// TIA Portal project "2022.06.10_多路模拟输入输出" (V17)

(* hardware
DEVICE "S7-1200 station_1"  S7-1200 Station
   slot 0: "Rack_0"  S7-1200 Rack  Rack  V1.0
   slot 1: "PLC_1"  CPU 1212C DC/DC/DC  6ES7 212-1AE40-0XB0  V4.5
   slot 2: "AI 4x13BIT/AQ 2x14BIT_1"  SM 1234 AI4/AQ2  6ES7 234-4HE30-0XB0  V1.0
*)

// ===== PLC "PLC_1"  CPU 1212C DC/DC/DC =====

VAR_GLOBAL   // PLC tag table "默认变量表"
   "所需频率" AT %IW96 : Word;
   "百分比" AT %MD40 : DWord;
   "模拟量输出通道" AT %MD44 : UDInt;
   "所需频率(1)" AT %MD0 : Real;
   "压力2模拟输入通道" AT %IW100 : Int;
   "压力2" AT %MD4 : Real;
END_VAR

FUNCTION "模拟量输入" : Void   // FC1, LAD
{ S7_Optimized_Access := 'TRUE' }
VERSION : 0.1
   VAR_INPUT
      模拟量输入上限 : Int;
      模拟量输入下限 : Int;
      工程之上限 : Real;
      工程值下限 : Real;
      模拟量输入值 : Int;
   END_VAR
   VAR_OUTPUT
      实际工程值 : Real;
   END_VAR
   VAR_TEMP
      百分比 : Bool;
   END_VAR
BEGIN

REGION Network 1
   // out只是中转，用temp
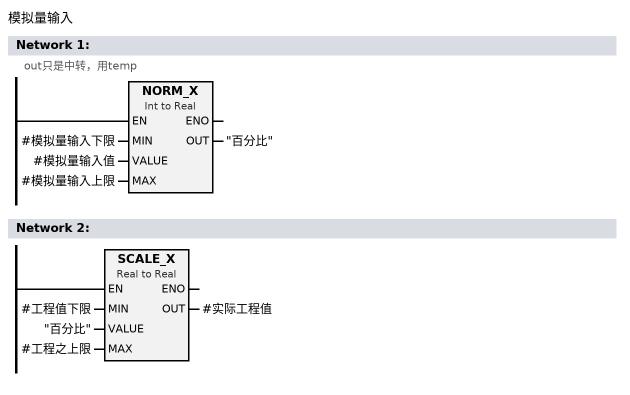
   RUNG wire#powerrail
      { S7_Templates := "[SrcType := Int, DestType := Real]" } Normalize(min := #模拟量输入下限, value := #模拟量输入值, max := #模拟量输入上限, out => "百分比")
   END_RUNG
   // the same network as SCL:
   "百分比" := NORM_X(MIN := #模拟量输入下限, VALUE := #模拟量输入值, MAX := #模拟量输入上限);
END_REGION

REGION Network 2
   RUNG wire#powerrail
      { S7_Templates := "[SrcType := Real, DestType := Real]" } Scale(min := #工程值下限, value := "百分比", max := #工程之上限, out => #实际工程值)
   END_RUNG
   // the same network as SCL:
   #实际工程值 := SCALE_X(MIN := #工程值下限, VALUE := "百分比", MAX := #工程之上限);
END_REGION
END_FUNCTION

FUNCTION "多路模拟量" : Void   // FC2, LAD
{ S7_Optimized_Access := 'TRUE' }
VERSION : 0.1
BEGIN

REGION Network 1
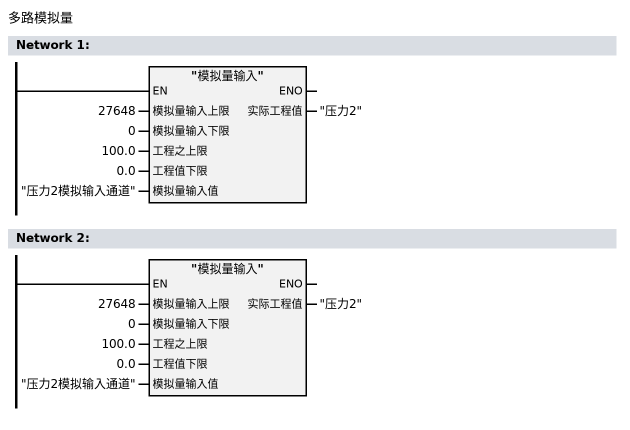
   RUNG wire#powerrail
      "模拟量输入"(模拟量输入上限 := 27648, 模拟量输入下限 := 0, 工程之上限 := 100.0, 工程值下限 := 0.0, 模拟量输入值 := "压力2模拟输入通道", 实际工程值 => "压力2")
   END_RUNG
   // the same network as SCL:
   "模拟量输入"(模拟量输入上限 := 27648, 模拟量输入下限 := 0, 工程之上限 := 100.0, 工程值下限 := 0.0, 模拟量输入值 := "压力2模拟输入通道", 实际工程值 => "压力2");
END_REGION

REGION Network 2
   RUNG wire#powerrail
      "模拟量输入"(模拟量输入上限 := 27648, 模拟量输入下限 := 0, 工程之上限 := 100.0, 工程值下限 := 0.0, 模拟量输入值 := "压力2模拟输入通道", 实际工程值 => "压力2")
   END_RUNG
   // the same network as SCL:
   "模拟量输入"(模拟量输入上限 := 27648, 模拟量输入下限 := 0, 工程之上限 := 100.0, 工程值下限 := 0.0, 模拟量输入值 := "压力2模拟输入通道", 实际工程值 => "压力2");
END_REGION
END_FUNCTION

ORGANIZATION_BLOCK "Main"   // OB1, LAD, ProgramCycle
TITLE = "Main Program Sweep (Cycle)"
{ S7_Optimized_Access := 'TRUE' }
VERSION : 0.1
   VAR_INPUT
      Initial_Call : Bool;   // Initial call of this OB
      Remanence : Bool;   // =True, if remanent data are available
   END_VAR
BEGIN

REGION Network 1
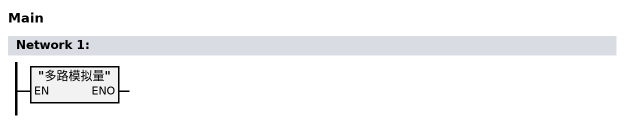
   RUNG wire#powerrail
      "多路模拟量"()
   END_RUNG
   // the same network as SCL:
   "多路模拟量"();
END_REGION
END_ORGANIZATION_BLOCK